(* Logix 5000 project; controller cal1615 1756-L62 rev 20.19; software revision 20.05; part 42 of 82 *)
(* tags used below, declared in another part *)
   FAULT : BOOL;   // Fault AFI
   p01r02_plc_scan_time_in_sec : REAL;   // System PLC Scan Time in Seconds
   p01r09 : routine;   // System Modes
   p01r09_pb_global_reset : BOOL;   // System Modes PB: Global Fault Reset
   p01r12_master_ramped_speed : REAL;   // System Line Accel Decel Control Master Ramped Speed
   p01r13_line_running : BOOL;   // System Line Start Sequence Line Running
   p01r13_line_slow_ramp : BOOL;   // System Line Start Sequence Start Line to Slow Speed
   p01r13_permissive_drives : BOOL;   // System Line Start Sequence Permissive Drives
   p20_ai_lc01 : REAL;   // Letoff Analog Input Line Tension Load Cell Splicer
   p20_ai_letoff_dia : REAL;   // Letoff Analog Inputs Letoff Roll Diameter [in]
   p20_ai_lob_speed : REAL;   // Letoff Inputs Letoff A Speed
   p20_ao_lob_selected_speed : REAL;   // Letoff Letoff B VFD Selected Speed
   p20_ao_lob_torque : REAL;
   p20_di_loa_active : BOOL;   // Letoff Digital Input Letoff A Active
   p20_di_loa_brake : BOOL;   // Letoff Input Letoff A Brake Temperature Ok
   p20_di_loa_temp : BOOL;   // Letoff Input Letoff A Motor Temperature Ok
   p20_di_lob_brake_thermostat : BOOL;   // Letoff Input Letoff B Brake Temperature OK
   p20_di_lob_fwd_dir : BOOL;   // Letoff Digital Inputs PB: Letoff B Jog FWD
   p20_di_lob_jog : BOOL;   // Letoff Digital Inputs PB: Letoff B Jog REV
   p20_di_lob_motor_thermostat : BOOL;   // Letoff Input Letoff B Motor Temperature Ok
   p20_di_lob_start : BOOL;   // Letoff Digital Input PB: Letoff B Start
   p20_di_lob_stop : BOOL;   // Letoff Digital Input PB: Letoff B Stop
   p20_do_close_nip : BOOL;   // Letoff Digital Output Feedroll Roll Nip Close
   p20_param_high_accel_rate : REAL;
   p20_param_high_decel_rate : REAL;
   p20_param_jog_accel_rate : REAL;
   p20_param_jog_decel_rate : REAL;
   p20_param_letoff_jog_speed : REAL;
   p20_param_lof_fast_fill : REAL;
   p20_param_lof_slow_fill : REAL;
   p20_param_lof_stop_fill : REAL;
   p20_param_norm_accel_rate : REAL;
   p20_param_norm_decel_rate : REAL;   // Letoff Parameter Letoff A Decel Rate
   p20_param_run_torque : REAL;
   p20_vfd_di_loa : acs800_di_normal;   // Letoff A VFD Inputs
   p20_vfd_di_lob : acs800_di_normal;   // Letoff B VFD Inputs
   p20_vfd_do_lob : acs800_do_normal;   // Letoff B VFD Outputs
   p20r10_speed_offset : REAL;   // Letoff Letoff Speed Control Speed Offset
   p20r13_state : DINT;   // Letoff Accumulator State
   p20r15 : routine;   // Letoff Letoff A VFD
   p20r15_request_tension : BOOL;   // Letoff Letoff A VFD Request Tension
   p20r15_timer_fault : TIMER[10];   // Letoff Letoff A VFD Fault Timer
   p20r15_timer_warning : TIMER[5];   // Letoff Letoff A VFD Warning Dwell Timer
   p20r16 : routine;   // Letoff Letoff B VFD
   p20r16_loa_accel_decel_ramp : SYS_ACC_DEC_RAMP;   // Letoff Letoff B VFD Accel/Decel Ramp
   p20r16_lob_accel : REAL;   // Letoff Letoff B VFD Accel Rate
   p20r16_lob_decel : REAL;   // Letoff Letoff B VFD Decel Rate
   p20r16_lob_on : BOOL;   // Letoff Letoff B On
   p20r16_lob_selected_speed : REAL;   // Letoff Letoff B VFD Selected Speed
   p20r16_permissive_run : BOOL;   // Letoff Letoff B VFD Permissive Run
   p20r16_request_jog_fwd : BOOL;   // Letoff Letoff B VFD Request Jog FWD
   p20r16_request_jog_rev : BOOL;   // Letoff Letoff B VFD Request Jog REV
   p20r16_request_over_speed : BOOL;   // Letoff Letoff B VFD Request Over Speed
   p20r16_request_position : BOOL;   // Letoff Letoff B VFD Request Position
   p20r16_request_stop : BOOL;   // Letoff Letoff B VFD Request Stop
   p20r16_request_tension : BOOL;   // Letoff Letoff B VFD Request Tension
   p20r16_request_thread_fwd : BOOL;
   p20r16_request_thread_rev : BOOL;
   p20r16_timer_fault : TIMER[10];   // Letoff Letoff B VFD Fault Dwell Timer
   p20r16_timer_warning : TIMER[4];   // Letoff Letoff B VFD Warning Dwell Timer
   p20r16_zero_speed : BOOL;   // Letoff Letoff B VFD Zero Speed
   p20r17 : routine;   // Letoff Letoff Diameter Calc
   p20r17_ave_control : CONTROL;   // Letoff Letoff Diameter Calc Average Control
   p20r17_diameter_clac_active : BOOL;   // Letoff Letoff Diameter Calc Active
   p20r17_letoff_avg_diam_inch : REAL;   // Letoff Letoff Diameter Calc Average Diameter [in]
   p20r17_letoff_diam_avg_stack : REAL[20];   // Letoff Letoff Diameter Calc Average Stack
   p20r17_stack_ctrl : CONTROL;   // Letoff Letoff Diameter Calc Stack Control
   p20r17_timer : TIMER[5];   // Letoff Letoff Diameter Calc Timer
   p20r17_timer_fault : TIMER[5];   // Letoff Letoff Diameter Calc Fault Dwell Timer
   p20r17_timer_warning : TIMER[5];   // Letoff Letoff Diameter Calc Warning Dwell Timer
   p20r17_winder_a_unload : REAL;   // Letoff Letoff Diameter Calc Temp Unload
   p20r18_index_complete : BOOL;   // Letoff Letoff Turret VFD Index Complete
   P21r01 : routine;
   p22_ao_selected_speed : REAL;   // Tension Stand 1 VFD Selected Speed
   p22r11_request_thread_fwd : BOOL;   // Tension Stand 1 VFD Request Thread FWD
   p22r11_request_thread_rev : BOOL;   // Tension Stand 1 VFD Request Thread REV
   p25r11_request_thread_fwd : BOOL;   // Tension Stand 2 VFD Request Thread FWD
   p25r11_request_thread_rev : BOOL;   // Tension Stand 2 VFD Request Thread REV
   p27r01 : routine;   // Winder Main
(* P20_Letoff, continued *)

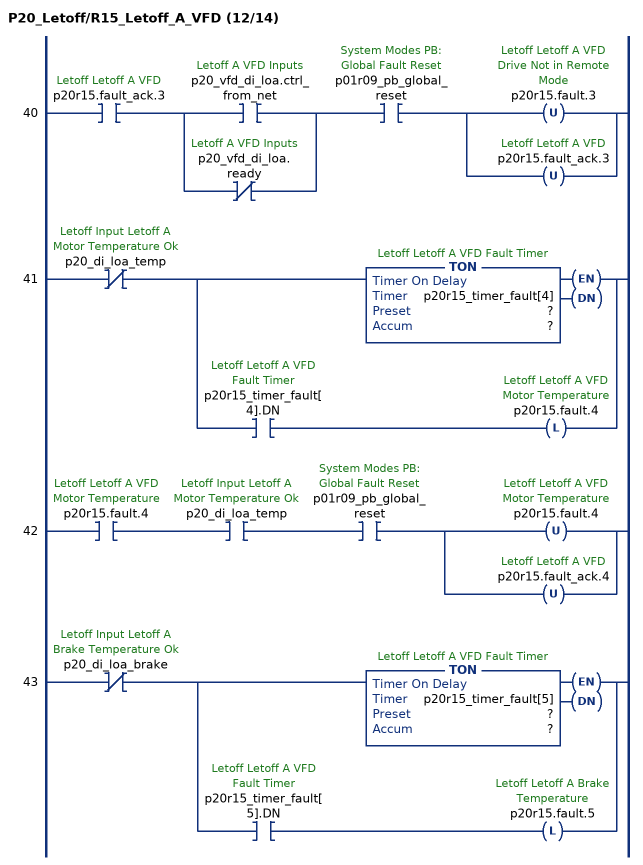
   [picture p791: P20_Letoff/R15_Letoff_A_VFD rungs 40-43]
   40: XIC(p20r15.fault_ack.3)[XIC(p20_vfd_di_loa.ctrl_from_net) ,XIO(p20_vfd_di_loa.ready) ]XIC(p01r09_pb_global_reset)[OTU(p20r15.fault.3) ,OTU(p20r15.fault_ack.3) ];
   41: XIO(p20_di_loa_temp)[TON(p20r15_timer_fault[4],?,?) ,XIC(p20r15_timer_fault[4].DN) OTL(p20r15.fault.4) ];
   42: XIC(p20r15.fault.4)XIC(p20_di_loa_temp)XIC(p01r09_pb_global_reset)[OTU(p20r15.fault.4) ,OTU(p20r15.fault_ack.4) ];
   43: XIO(p20_di_loa_brake)[TON(p20r15_timer_fault[5],?,?) ,XIC(p20r15_timer_fault[5].DN) OTL(p20r15.fault.5) ];
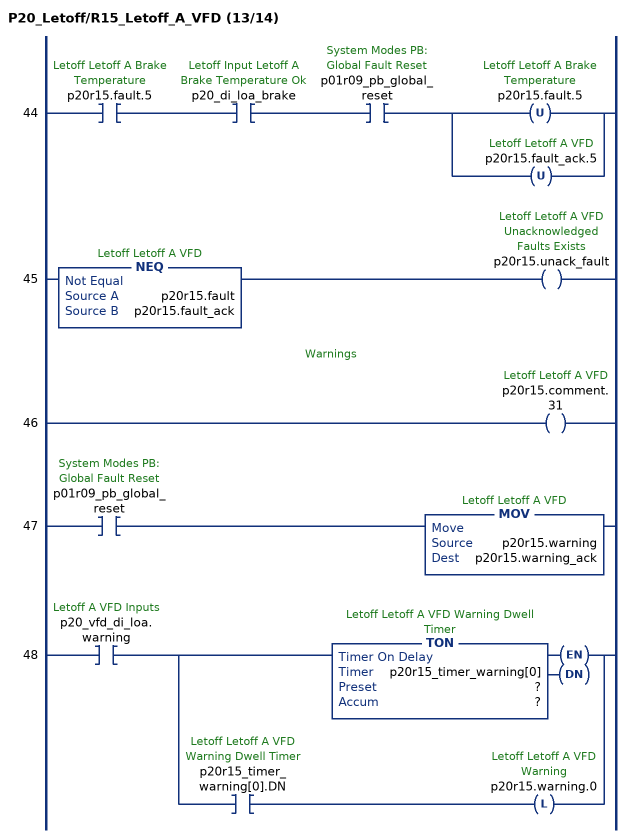
   44: XIC(p20r15.fault.5)XIC(p20_di_loa_brake)XIC(p01r09_pb_global_reset)[OTU(p20r15.fault.5) ,OTU(p20r15.fault_ack.5) ];
   45: NEQ(p20r15.fault,p20r15.fault_ack)OTE(p20r15.unack_fault);
   // Warnings
   46: OTE(p20r15.comment.31);
   47: XIC(p01r09_pb_global_reset)MOV(p20r15.warning,p20r15.warning_ack);
   48: XIC(p20_vfd_di_loa.warning)[TON(p20r15_timer_warning[0],?,?) ,XIC(p20r15_timer_warning[0].DN) OTL(p20r15.warning.0) ];
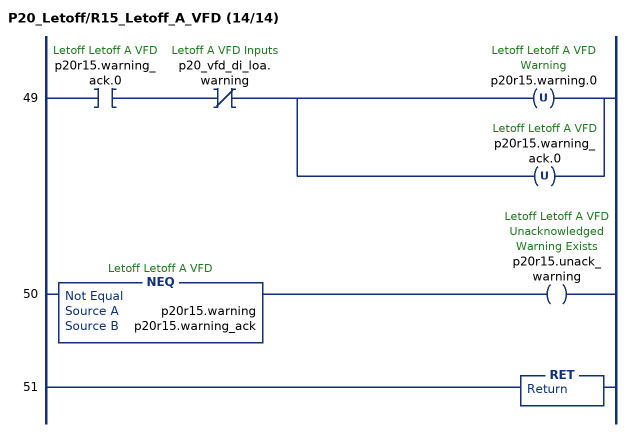
   49: XIC(p20r15.warning_ack.0)XIO(p20_vfd_di_loa.warning)[OTU(p20r15.warning.0) ,OTU(p20r15.warning_ack.0) ];
   50: NEQ(p20r15.warning,p20r15.warning_ack)OTE(p20r15.unack_warning);
   51: RET();
END_ROUTINE

ROUTINE R16_Letoff_B_VFD   (* ladder *)
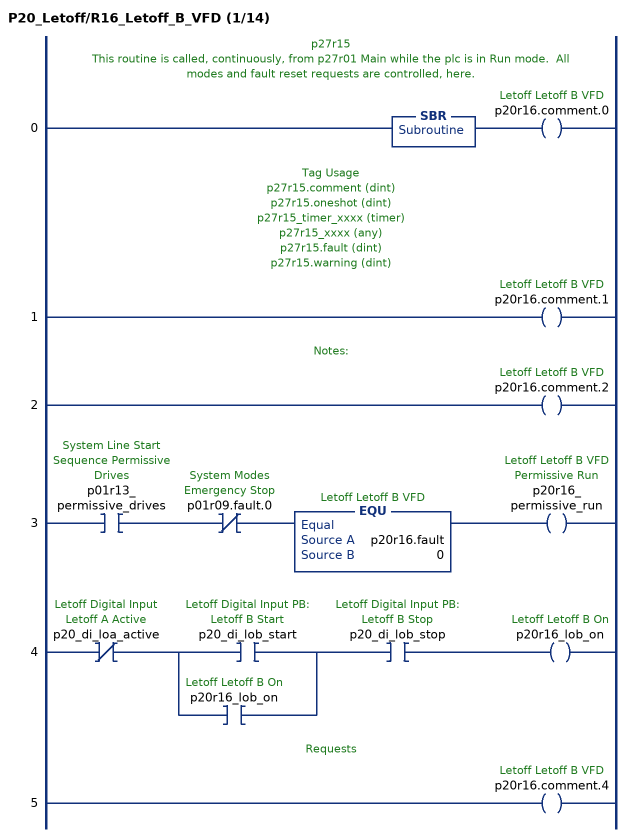
   // p27r15
   // This routine is called, continuously, from p27r01 Main while the plc is in Run mode.  All modes and fault reset requests are controlled, here.
   0: SBR()OTE(p20r16.comment.0);
   // Tag Usage
   // p27r15.comment (dint)
   // p27r15.oneshot (dint)
   // p27r15_timer_xxxx (timer)
   // p27r15_xxxx (any)
   // p27r15.fault (dint)
   // p27r15.warning (dint)
   1: OTE(p20r16.comment.1);
   // Notes:
   2: OTE(p20r16.comment.2);
   3: XIC(p01r13_permissive_drives)XIO(p01r09.fault.0)EQU(p20r16.fault,0)OTE(p20r16_permissive_run);
   4: XIO(p20_di_loa_active)[XIC(p20_di_lob_start) ,XIC(p20r16_lob_on) ]XIC(p20_di_lob_stop)OTE(p20r16_lob_on);
   // Requests
   5: OTE(p20r16.comment.4);
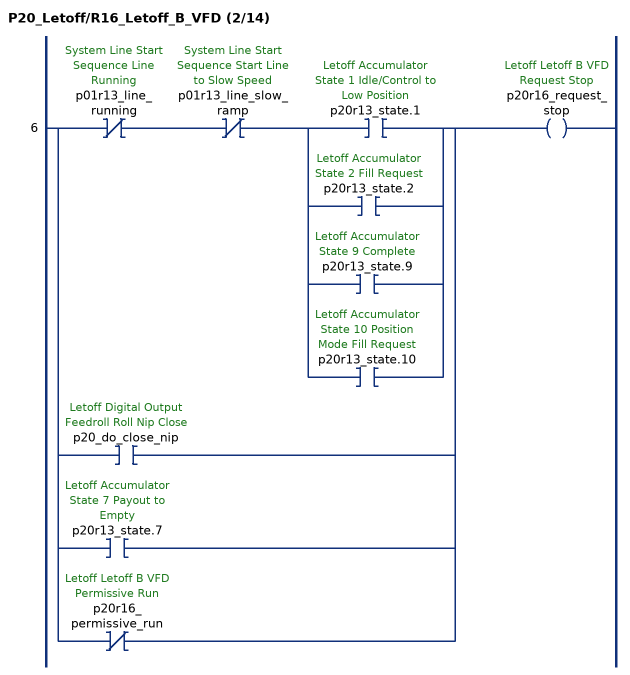
   6: [XIO(p01r13_line_running) XIO(p01r13_line_slow_ramp) [XIC(p20r13_state.1) ,XIC(p20r13_state.2) ,XIC(p20r13_state.9) ,XIC(p20r13_state.10) ] ,XIC(p20_do_close_nip) ,XIC(p20r13_state.7) ,XIO(p20r16_permissive_run) ]OTE(p20r16_request_stop);
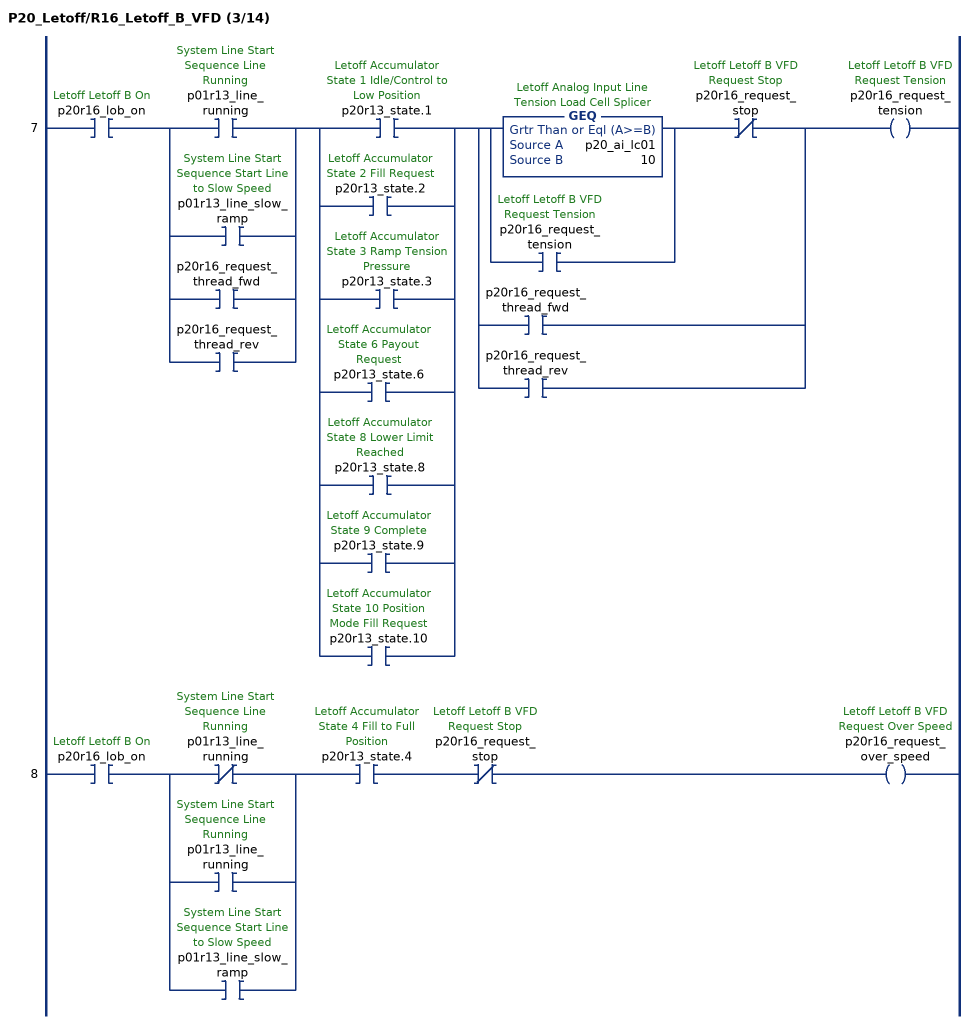
   7: XIC(p20r16_lob_on)[XIC(p01r13_line_running) ,XIC(p01r13_line_slow_ramp) ,XIC(p20r16_request_thread_fwd) ,XIC(p20r16_request_thread_rev) ][XIC(p20r13_state.1) ,XIC(p20r13_state.2) ,XIC(p20r13_state.3) ,XIC(p20r13_state.6) ,XIC(p20r13_state.8) ,XIC(p20r13_state.9) ,XIC(p20r13_state.10) ][[GEQ(p20_ai_lc01,10) ,XIC(p20r16_request_tension) ] XIO(p20r16_request_stop) ,XIC(p20r16_request_thread_fwd) ,XIC(p20r16_request_thread_rev) ]OTE(p20r16_request_tension);
   8: XIC(p20r16_lob_on)[XIO(p01r13_line_running) ,XIC(p01r13_line_running) ,XIC(p01r13_line_slow_ramp) ]XIC(p20r13_state.4)XIO(p20r16_request_stop)OTE(p20r16_request_over_speed);
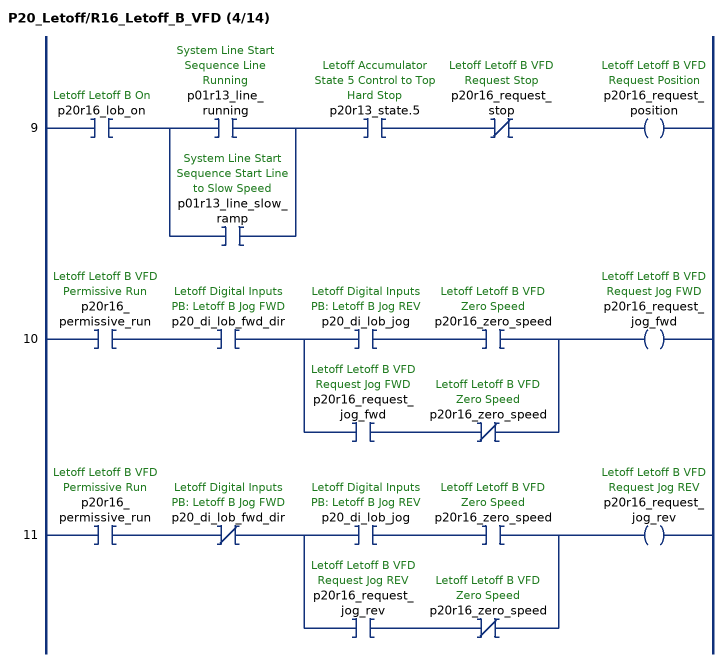
   9: XIC(p20r16_lob_on)[XIC(p01r13_line_running) ,XIC(p01r13_line_slow_ramp) ]XIC(p20r13_state.5)XIO(p20r16_request_stop)OTE(p20r16_request_position);
   10: XIC(p20r16_permissive_run)XIC(p20_di_lob_fwd_dir)[XIC(p20_di_lob_jog) XIC(p20r16_zero_speed) ,XIC(p20r16_request_jog_fwd) XIO(p20r16_zero_speed) ]OTE(p20r16_request_jog_fwd);
   11: XIC(p20r16_permissive_run)XIO(p20_di_lob_fwd_dir)[XIC(p20_di_lob_jog) XIC(p20r16_zero_speed) ,XIC(p20r16_request_jog_rev) XIO(p20r16_zero_speed) ]OTE(p20r16_request_jog_rev);
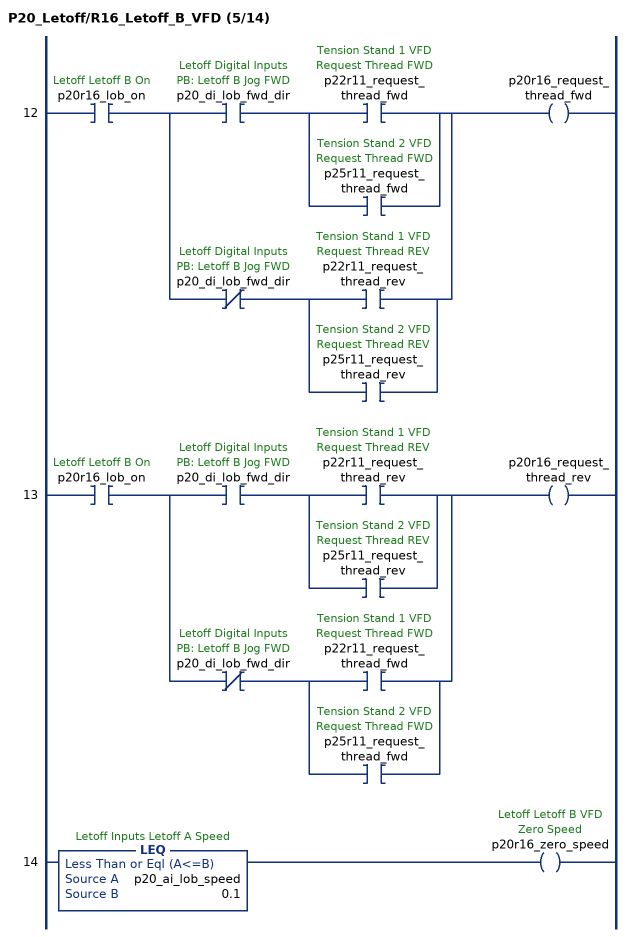
   12: XIC(p20r16_lob_on)[XIC(p20_di_lob_fwd_dir) [XIC(p22r11_request_thread_fwd) ,XIC(p25r11_request_thread_fwd) ] ,XIO(p20_di_lob_fwd_dir) [XIC(p22r11_request_thread_rev) ,XIC(p25r11_request_thread_rev) ] ]OTE(p20r16_request_thread_fwd);
   13: XIC(p20r16_lob_on)[XIC(p20_di_lob_fwd_dir) [XIC(p22r11_request_thread_rev) ,XIC(p25r11_request_thread_rev) ] ,XIO(p20_di_lob_fwd_dir) [XIC(p22r11_request_thread_fwd) ,XIC(p25r11_request_thread_fwd) ] ]OTE(p20r16_request_thread_rev);
   14: LEQ(p20_ai_lob_speed,0.1)OTE(p20r16_zero_speed);
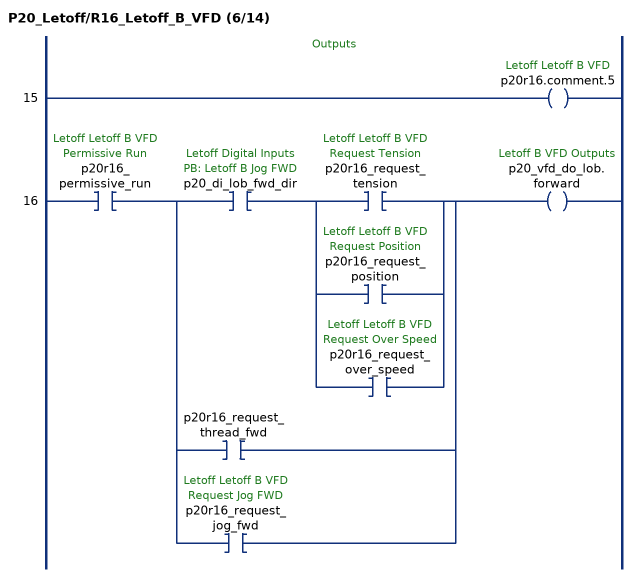
   // Outputs
   15: OTE(p20r16.comment.5);
   16: XIC(p20r16_permissive_run)[XIC(p20_di_lob_fwd_dir) [XIC(p20r16_request_tension) ,XIC(p20r16_request_position) ,XIC(p20r16_request_over_speed) ] ,XIC(p20r16_request_thread_fwd) ,XIC(p20r16_request_jog_fwd) ]OTE(p20_vfd_do_lob.forward);
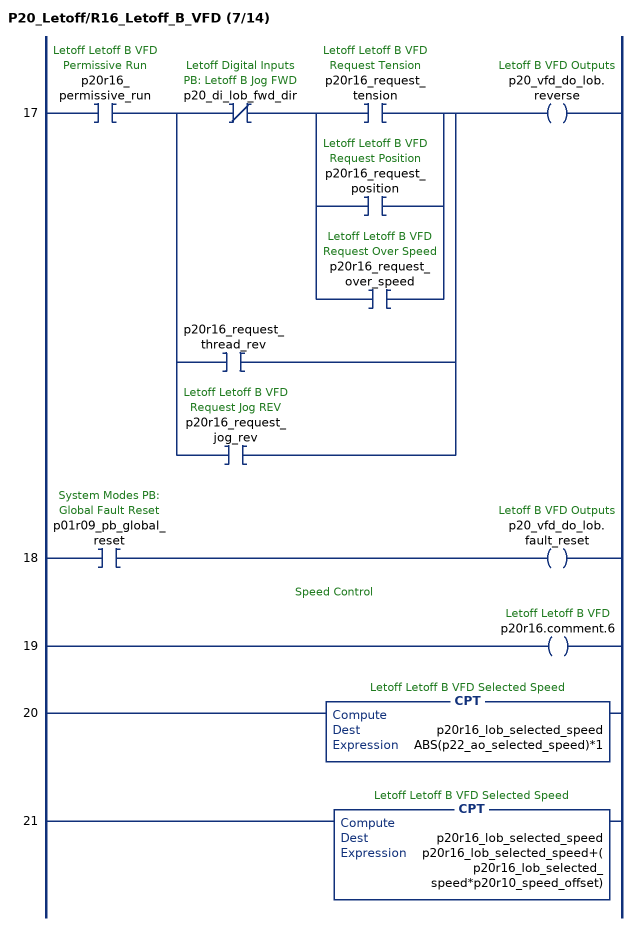
   17: XIC(p20r16_permissive_run)[XIO(p20_di_lob_fwd_dir) [XIC(p20r16_request_tension) ,XIC(p20r16_request_position) ,XIC(p20r16_request_over_speed) ] ,XIC(p20r16_request_thread_rev) ,XIC(p20r16_request_jog_rev) ]OTE(p20_vfd_do_lob.reverse);
   18: XIC(p01r09_pb_global_reset)OTE(p20_vfd_do_lob.fault_reset);
   // Speed Control
   19: OTE(p20r16.comment.6);
   20: CPT(p20r16_lob_selected_speed,ABS(p22_ao_selected_speed)*1);
   21: CPT(p20r16_lob_selected_speed,p20r16_lob_selected_speed+(p20r16_lob_selected_speed*p20r10_speed_offset));
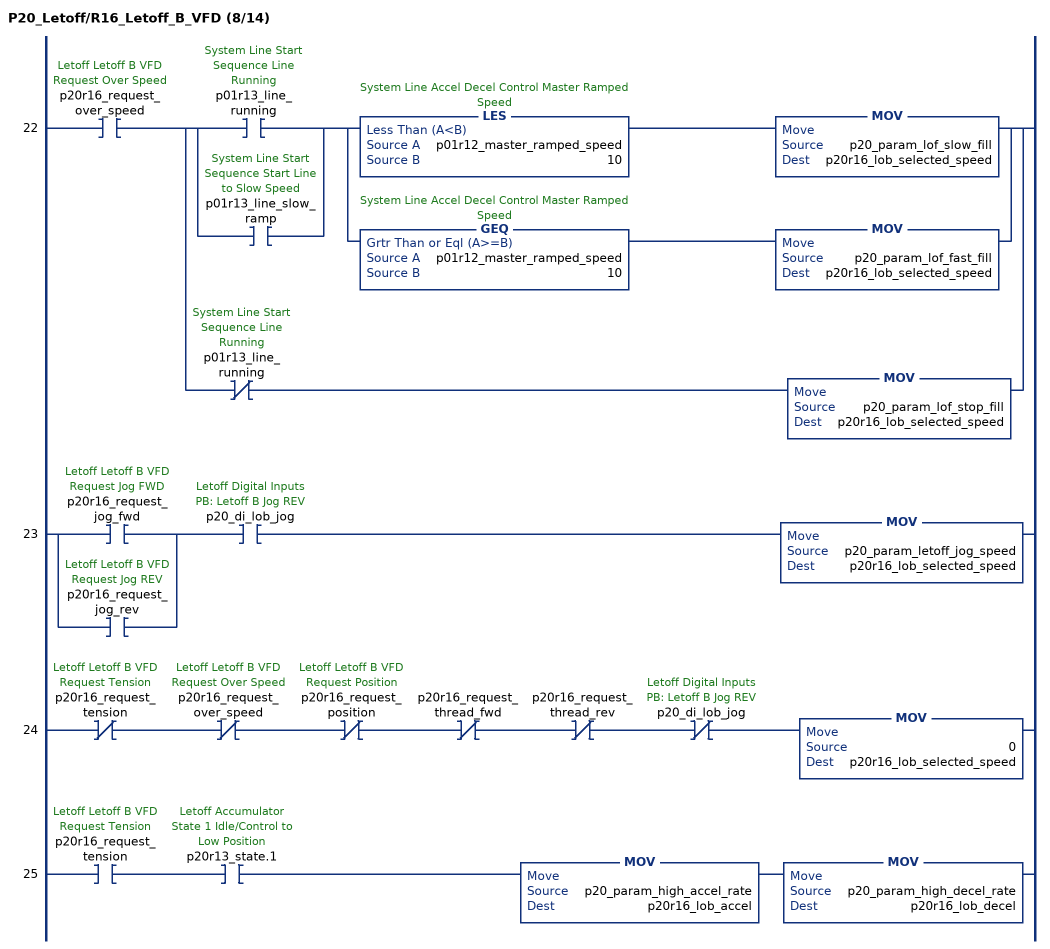
   22: XIC(p20r16_request_over_speed)[[XIC(p01r13_line_running) ,XIC(p01r13_line_slow_ramp) ] [LES(p01r12_master_ramped_speed,10) MOV(p20_param_lof_slow_fill,p20r16_lob_selected_speed) ,GEQ(p01r12_master_ramped_speed,10) MOV(p20_param_lof_fast_fill,p20r16_lob_selected_speed) ] ,XIO(p01r13_line_running) MOV(p20_param_lof_stop_fill,p20r16_lob_selected_speed) ];
   23: [XIC(p20r16_request_jog_fwd) ,XIC(p20r16_request_jog_rev) ]XIC(p20_di_lob_jog)MOV(p20_param_letoff_jog_speed,p20r16_lob_selected_speed);
   24: XIO(p20r16_request_tension)XIO(p20r16_request_over_speed)XIO(p20r16_request_position)XIO(p20r16_request_thread_fwd)XIO(p20r16_request_thread_rev)XIO(p20_di_lob_jog)MOV(0,p20r16_lob_selected_speed);
   25: XIC(p20r16_request_tension)XIC(p20r13_state.1)MOV(p20_param_high_accel_rate,p20r16_lob_accel)MOV(p20_param_high_decel_rate,p20r16_lob_decel);
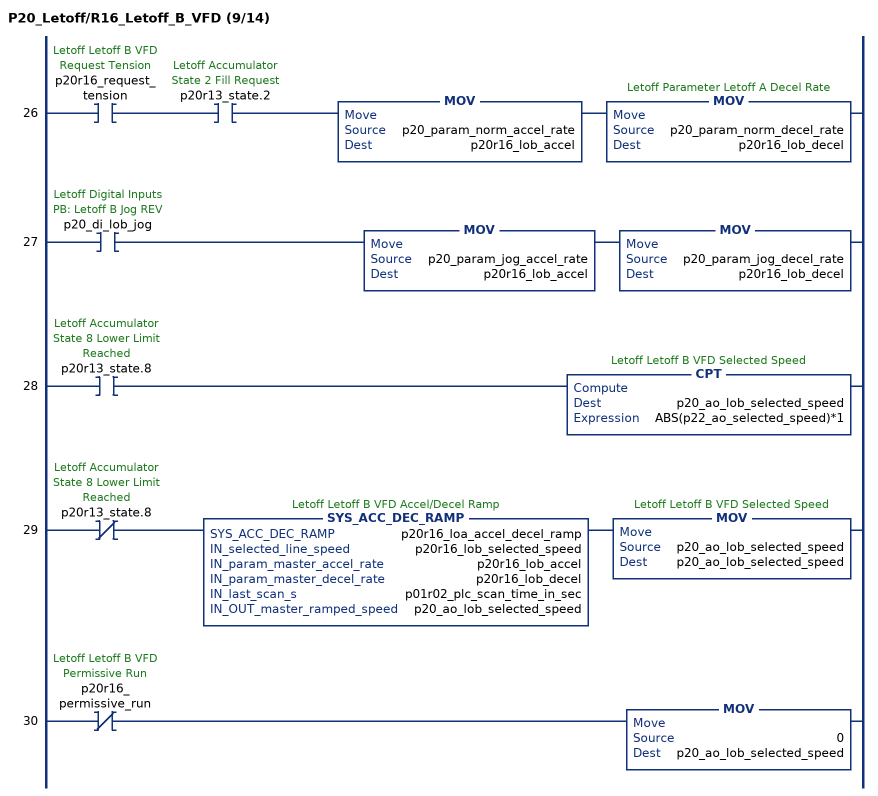
   26: XIC(p20r16_request_tension)XIC(p20r13_state.2)MOV(p20_param_norm_accel_rate,p20r16_lob_accel)MOV(p20_param_norm_decel_rate,p20r16_lob_decel);
   27: XIC(p20_di_lob_jog)MOV(p20_param_jog_accel_rate,p20r16_lob_accel)MOV(p20_param_jog_decel_rate,p20r16_lob_decel);
   28: XIC(p20r13_state.8)CPT(p20_ao_lob_selected_speed,ABS(p22_ao_selected_speed)*1);
   29: XIO(p20r13_state.8)SYS_ACC_DEC_RAMP(p20r16_loa_accel_decel_ramp,p20r16_lob_selected_speed,p20r16_lob_accel,p20r16_lob_decel,p01r02_plc_scan_time_in_sec,p20_ao_lob_selected_speed)MOV(p20_ao_lob_selected_speed,p20_ao_lob_selected_speed);
   30: XIO(p20r16_permissive_run)MOV(0,p20_ao_lob_selected_speed);
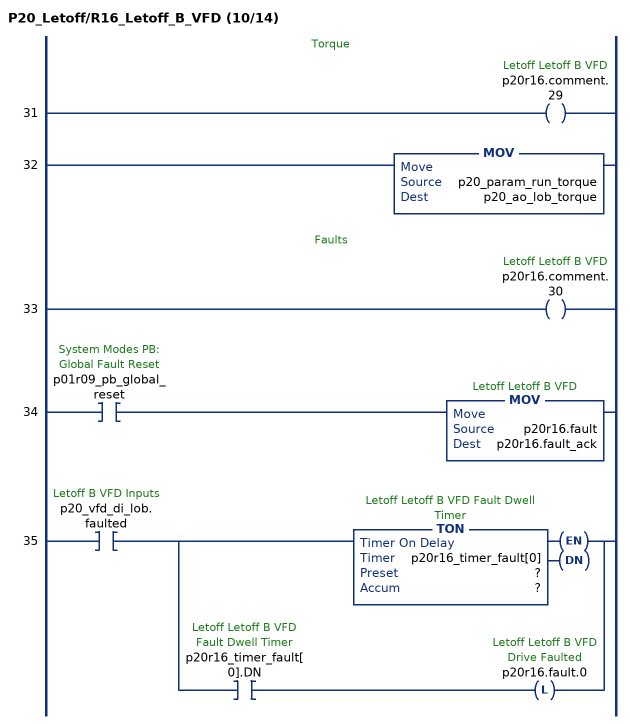
   // Torque
   31: OTE(p20r16.comment.29);
   32: MOV(p20_param_run_torque,p20_ao_lob_torque);
   // Faults
   33: OTE(p20r16.comment.30);
   34: XIC(p01r09_pb_global_reset)MOV(p20r16.fault,p20r16.fault_ack);
   35: XIC(p20_vfd_di_lob.faulted)[TON(p20r16_timer_fault[0],?,?) ,XIC(p20r16_timer_fault[0].DN) OTL(p20r16.fault.0) ];
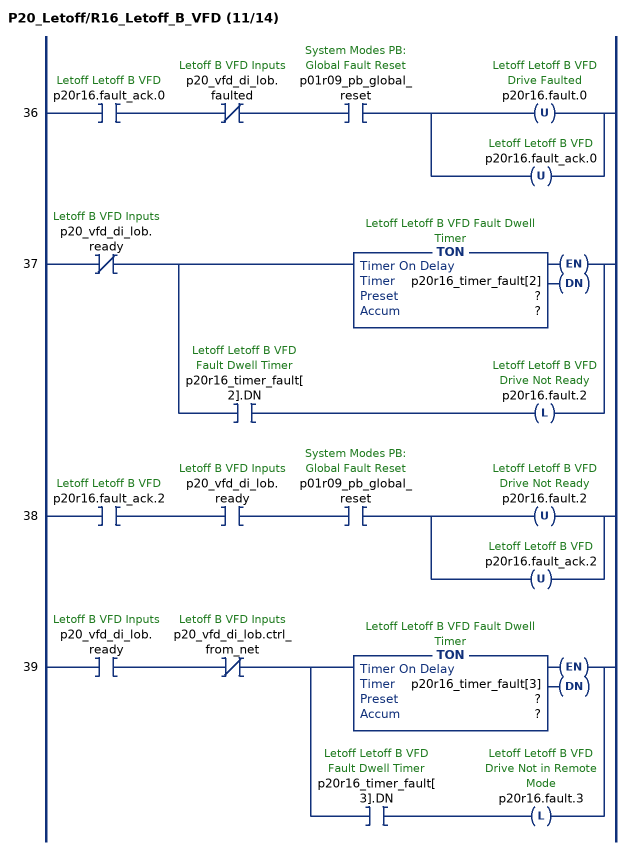
   36: XIC(p20r16.fault_ack.0)XIO(p20_vfd_di_lob.faulted)XIC(p01r09_pb_global_reset)[OTU(p20r16.fault.0) ,OTU(p20r16.fault_ack.0) ];
   37: XIO(p20_vfd_di_lob.ready)[TON(p20r16_timer_fault[2],?,?) ,XIC(p20r16_timer_fault[2].DN) OTL(p20r16.fault.2) ];
   38: XIC(p20r16.fault_ack.2)XIC(p20_vfd_di_lob.ready)XIC(p01r09_pb_global_reset)[OTU(p20r16.fault.2) ,OTU(p20r16.fault_ack.2) ];
   39: XIC(p20_vfd_di_lob.ready)XIO(p20_vfd_di_lob.ctrl_from_net)[TON(p20r16_timer_fault[3],?,?) ,XIC(p20r16_timer_fault[3].DN) OTL(p20r16.fault.3) ];
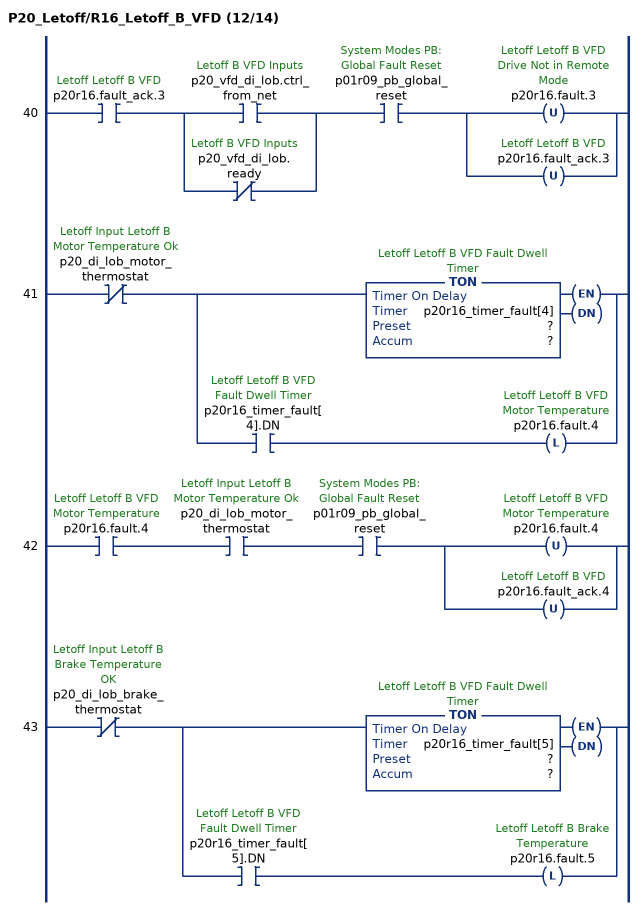
   40: XIC(p20r16.fault_ack.3)[XIC(p20_vfd_di_lob.ctrl_from_net) ,XIO(p20_vfd_di_lob.ready) ]XIC(p01r09_pb_global_reset)[OTU(p20r16.fault.3) ,OTU(p20r16.fault_ack.3) ];
   41: XIO(p20_di_lob_motor_thermostat)[TON(p20r16_timer_fault[4],?,?) ,XIC(p20r16_timer_fault[4].DN) OTL(p20r16.fault.4) ];
   42: XIC(p20r16.fault.4)XIC(p20_di_lob_motor_thermostat)XIC(p01r09_pb_global_reset)[OTU(p20r16.fault.4) ,OTU(p20r16.fault_ack.4) ];
   43: XIO(p20_di_lob_brake_thermostat)[TON(p20r16_timer_fault[5],?,?) ,XIC(p20r16_timer_fault[5].DN) OTL(p20r16.fault.5) ];
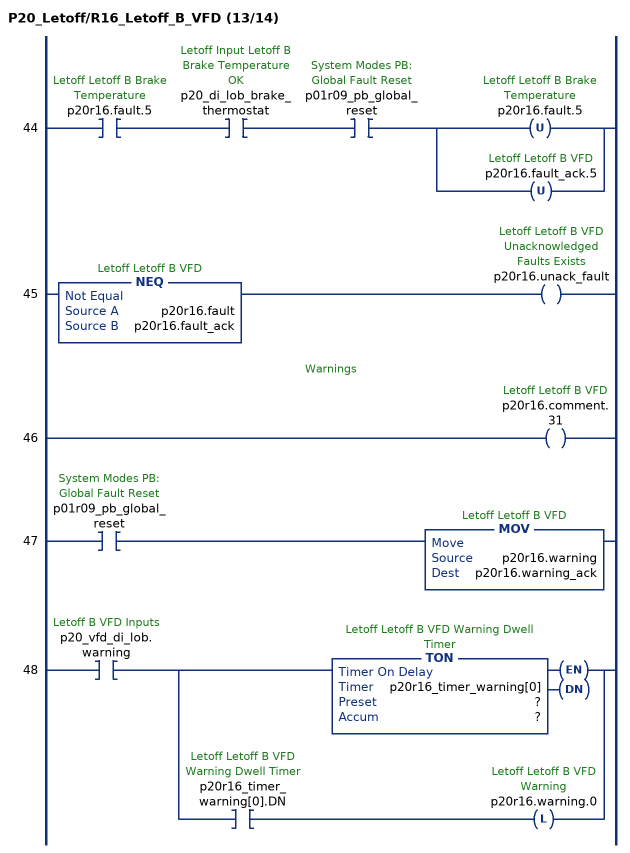
   44: XIC(p20r16.fault.5)XIC(p20_di_lob_brake_thermostat)XIC(p01r09_pb_global_reset)[OTU(p20r16.fault.5) ,OTU(p20r16.fault_ack.5) ];
   45: NEQ(p20r16.fault,p20r16.fault_ack)OTE(p20r16.unack_fault);
   // Warnings
   46: OTE(p20r16.comment.31);
   47: XIC(p01r09_pb_global_reset)MOV(p20r16.warning,p20r16.warning_ack);
   48: XIC(p20_vfd_di_lob.warning)[TON(p20r16_timer_warning[0],?,?) ,XIC(p20r16_timer_warning[0].DN) OTL(p20r16.warning.0) ];
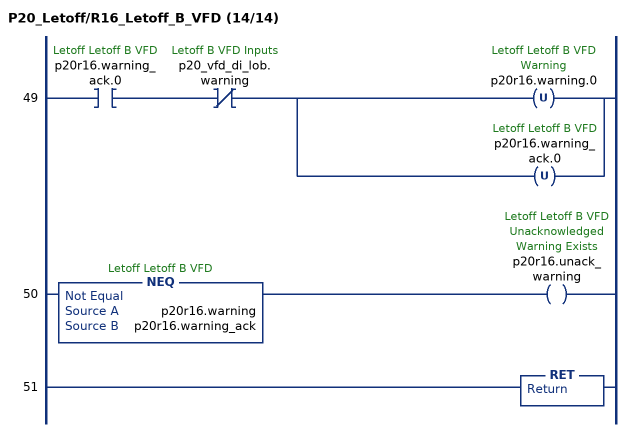
   49: XIC(p20r16.warning_ack.0)XIO(p20_vfd_di_lob.warning)[OTU(p20r16.warning.0) ,OTU(p20r16.warning_ack.0) ];
   50: NEQ(p20r16.warning,p20r16.warning_ack)OTE(p20r16.unack_warning);
   51: RET();
END_ROUTINE

ROUTINE R17_Letoff_Diameter_Calc   (* ladder *)
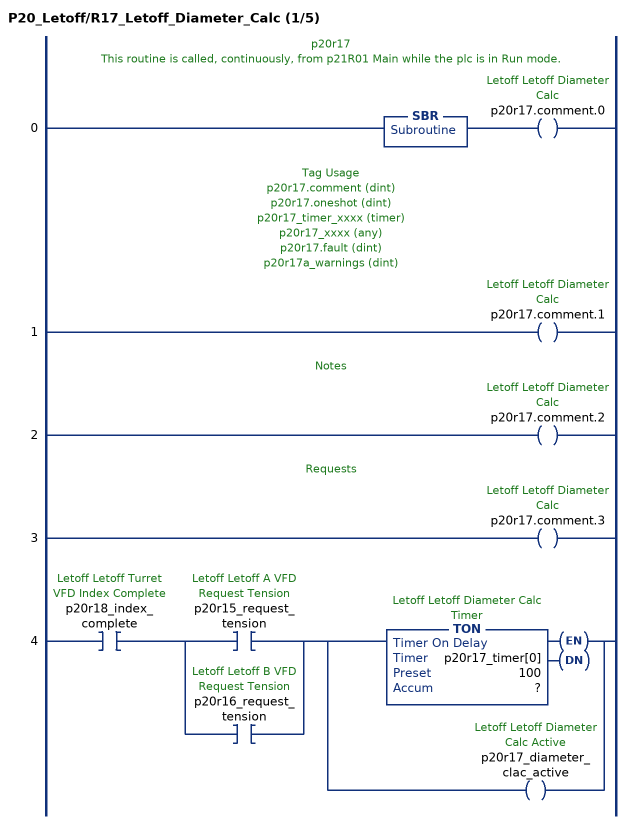
   // p20r17
   // This routine is called, continuously, from p21R01 Main while the plc is in Run mode.
   0: SBR()OTE(p20r17.comment.0);
   // Tag Usage
   // p20r17.comment (dint)
   // p20r17.oneshot (dint)
   // p20r17_timer_xxxx (timer)
   // p20r17_xxxx (any)
   // p20r17.fault (dint)
   // p20r17a_warnings (dint)
   1: OTE(p20r17.comment.1);
   // Notes
   2: OTE(p20r17.comment.2);
   // Requests
   3: OTE(p20r17.comment.3);
   4: XIC(p20r18_index_complete)[XIC(p20r15_request_tension) ,XIC(p20r16_request_tension) ][TON(p20r17_timer[0],?,?) ,OTE(p20r17_diameter_clac_active) ];
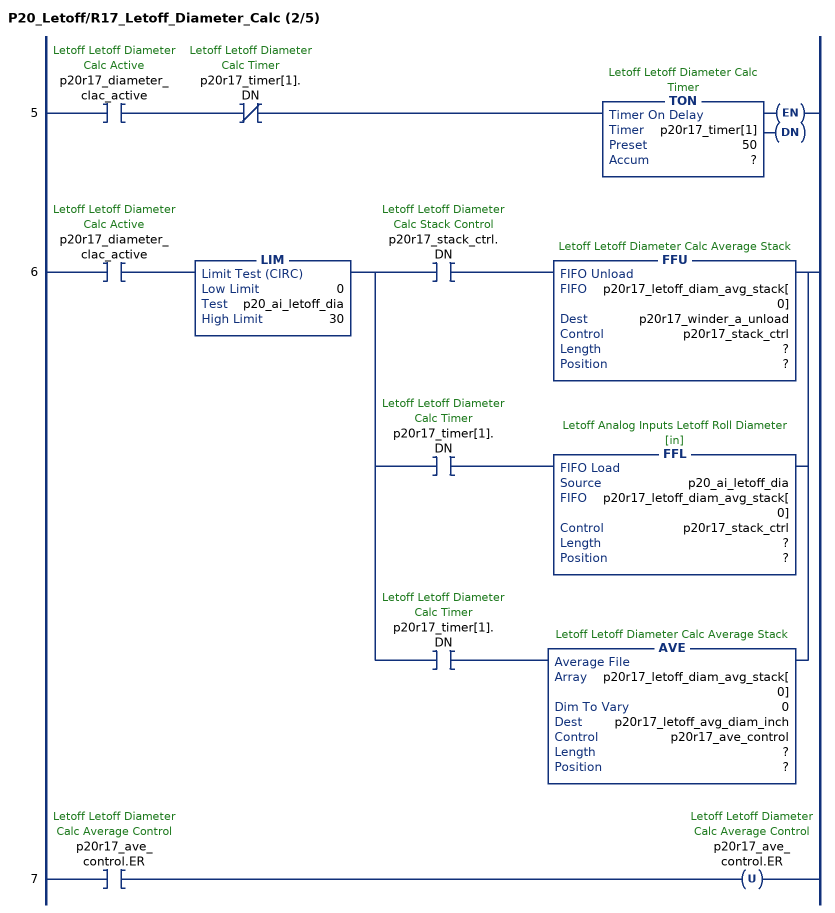
   5: XIC(p20r17_diameter_clac_active)XIO(p20r17_timer[1].DN)TON(p20r17_timer[1],?,?);
   6: XIC(p20r17_diameter_clac_active)LIM(0,p20_ai_letoff_dia,30)[XIC(p20r17_stack_ctrl.DN) FFU(p20r17_letoff_diam_avg_stack[0],p20r17_winder_a_unload,p20r17_stack_ctrl,?,?) ,XIC(p20r17_timer[1].DN) FFL(p20_ai_letoff_dia,p20r17_letoff_diam_avg_stack[0],p20r17_stack_ctrl,?,?) ,XIC(p20r17_timer[1].DN) AVE(p20r17_letoff_diam_avg_stack[0],0,p20r17_letoff_avg_diam_inch,p20r17_ave_control,?,?) ];
   7: XIC(p20r17_ave_control.ER)OTU(p20r17_ave_control.ER);
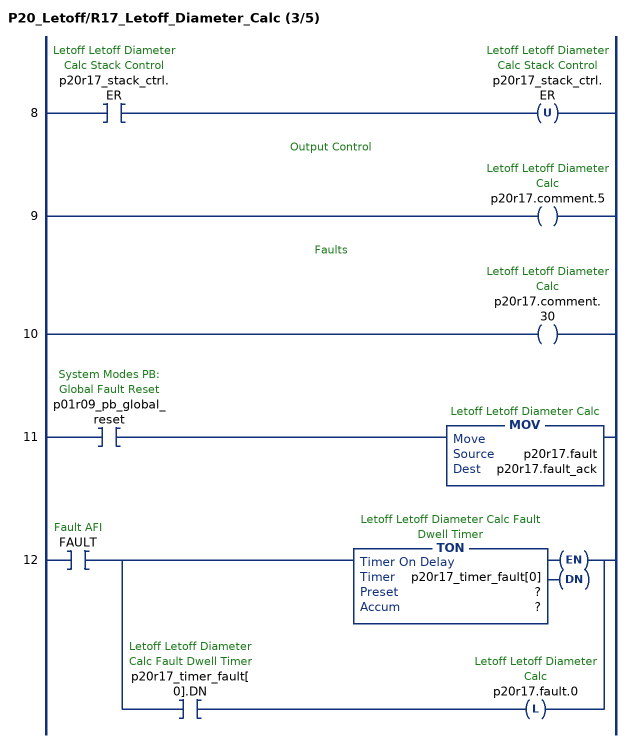
   8: XIC(p20r17_stack_ctrl.ER)OTU(p20r17_stack_ctrl.ER);
   // Output Control
   9: OTE(p20r17.comment.5);
   // Faults
   10: OTE(p20r17.comment.30);
   11: XIC(p01r09_pb_global_reset)MOV(p20r17.fault,p20r17.fault_ack);
   12: XIC(FAULT)[TON(p20r17_timer_fault[0],?,?) ,XIC(p20r17_timer_fault[0].DN) OTL(p20r17.fault.0) ];
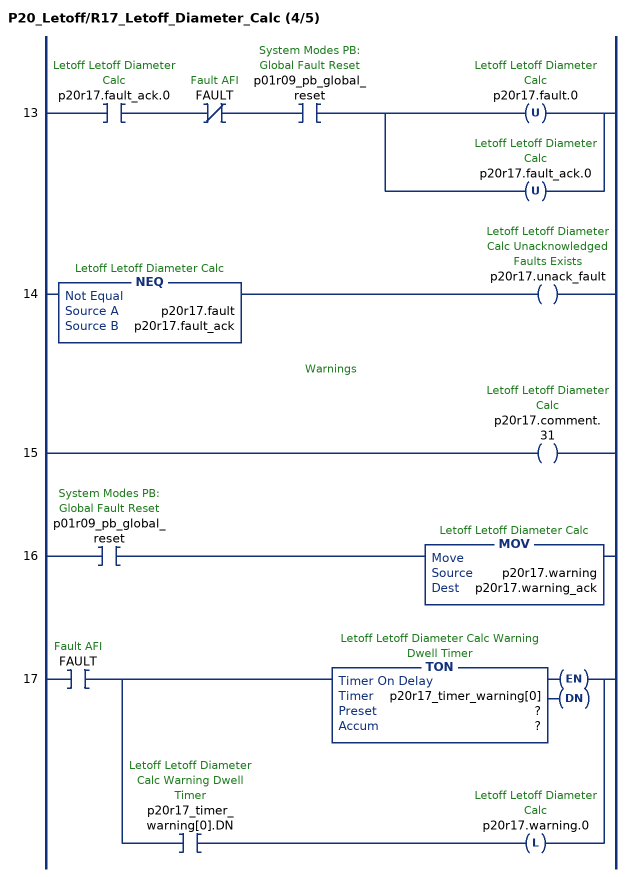
   13: XIC(p20r17.fault_ack.0)XIO(FAULT)XIC(p01r09_pb_global_reset)[OTU(p20r17.fault.0) ,OTU(p20r17.fault_ack.0) ];
   14: NEQ(p20r17.fault,p20r17.fault_ack)OTE(p20r17.unack_fault);
   // Warnings
   15: OTE(p20r17.comment.31);
   16: XIC(p01r09_pb_global_reset)MOV(p20r17.warning,p20r17.warning_ack);
   17: XIC(FAULT)[TON(p20r17_timer_warning[0],?,?) ,XIC(p20r17_timer_warning[0].DN) OTL(p20r17.warning.0) ];
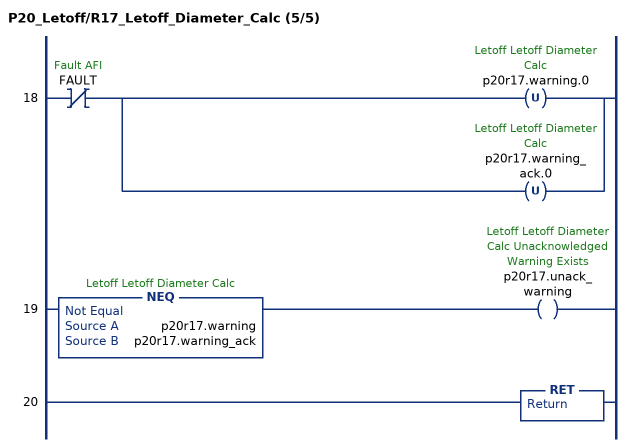
   18: XIO(FAULT)[OTU(p20r17.warning.0) ,OTU(p20r17.warning_ack.0) ];
   19: NEQ(p20r17.warning,p20r17.warning_ack)OTE(p20r17.unack_warning);
   20: RET();
END_ROUTINE
